Omron Sysmac Studio project Q14-16_2 (Sysmac Studio 1.23.0.14, StandardProject)

# Controller new_Controller_0: NX1P2-1040DT1 version 1.18
Task PrimaryTask (priority 4, period or condition 8000): Programa0

VAR_GLOBAL
    PP : BOOL;  (* at BuiltInIO://cpu/#0/Input_Bit_00 *)
    PM : BOOL;  (* at BuiltInIO://cpu/#0/Input_Bit_01 *)
    PR : BOOL;  (* at BuiltInIO://cpu/#0/Input_Bit_02 *)
    marcha_atras : BOOL;  (* at BuiltInIO://cpu/#0/Output_Bit_00 *)
    state : INT;
END_VAR
VAR_GLOBAL RETAIN
    rpm AT %D0 : DINT;  (* published *)
    mm_s AT %D4 : REAL;  (* published *)
END_VAR
VAR_GLOBAL
    Ch1Enable : BOOL;  (* at IOBus://unit#1/Ch1 Encoder Counter Operation Command/Ch1 Counter Enable *)
    Ch1Pulses : DINT;  (* at IOBus://unit#1/Ch1 Encoder Present Position *)
    Ch1PulseRate : UDINT;  (* at IOBus://unit#1/Ch1 Pulse Rate *)
    Ch1PeriodEnable : BOOL;  (* at IOBus://unit#1/Ch1 Pulse Period Measurement Function/Ch1 Pulse Period Measurement Enable *)
    detector_inicial : BOOL;  (* at BuiltInIO://cpu/#0/Input_Bit_03 *)
    marcha_adelante : BOOL;  (* at BuiltInIO://cpu/#0/Output_Bit_01 *)
END_VAR
VAR_GLOBAL RETAIN
    mm AT %D8 : DINT;  (* published *)
END_VAR
VAR_GLOBAL
    Ch1Reset : BOOL;  (* at IOBus://unit#1/Ch1 Encoder Counter Operation Command/Ch1 Internal Reset Execution *)
    multivelocidad_1 : BOOL;  (* at BuiltInIO://cpu/#0/Output_Bit_02 *)
    multivelocidad_2 : BOOL;  (* at BuiltInIO://cpu/#0/Output_Bit_03 *)
END_VAR
VAR_GLOBAL RETAIN
    selector_velocidad AT %D12 : INT;  (* published *)
    frecuencia_aplicada AT %D16 : INT;  (* published *)
    rpm_30hz AT %D20 : DINT;  (* published *)
    rpm_50hz AT %D24 : DINT;  (* published *)
    rpm_80hz AT %D28 : DINT;  (* published *)
    mm_s_30hz AT %D32 : REAL;  (* published *)
    mm_s_50hz AT %D36 : REAL;  (* published *)
    mm_s_80hz AT %D40 : REAL;  (* published *)
    MC_state AT %D7 : INT := 0;  (* published *)
END_VAR
VAR_GLOBAL
    PM_HMI AT %W0.00 : BOOL;  (* published *)
    PP_HMI AT %W0.01 : BOOL;  (* published *)
    PR_HMI AT %W0.02 : BOOL;  (* published *)
    PM_VAR : BOOL;
    PP_VAR : BOOL;
    PR_VAR : BOOL;
END_VAR
VAR_GLOBAL RETAIN
    deslizamiento AT %D44 : REAL;  (* published *)
END_VAR

PROGRAM Programa0
VAR CONSTANT
    time_window : INT := 500;
    encoder_resolution : INT := 8000;
END_VAR
VAR
    state : INT;
    velocidad_sincrona : REAL;
END_VAR
VAR_EXTERNAL
    Ch1Enable : BOOL;
    Ch1Pulses : DINT;
    rpm : DINT;
    Ch1PulseRate : UDINT;
    Ch1PeriodEnable : BOOL;
    PP : BOOL;
    PM : BOOL;
    detector_inicial : BOOL;
    marcha_adelante : BOOL;
    marcha_atras : BOOL;
    Ch1Reset : BOOL;
    PR : BOOL;
    mm : DINT;
    multivelocidad_1 : BOOL;
    multivelocidad_2 : BOOL;
    frecuencia_aplicada : INT;
    rpm_30hz : DINT;
    mm_s_30hz : REAL;
    rpm_50hz : DINT;
    mm_s_50hz : REAL;
    rpm_80hz : DINT;
    mm_s_80hz : REAL;
    selector_velocidad : INT;
    mm_s : REAL;
    PM_VAR : BOOL;
    PM_HMI : BOOL;
    PP_HMI : BOOL;
    PP_VAR : BOOL;
    PR_HMI : BOOL;
    PR_VAR : BOOL;
    deslizamiento : REAL;
END_VAR

(* Section calculos_encoder: ladder, written here as Structured Text *)

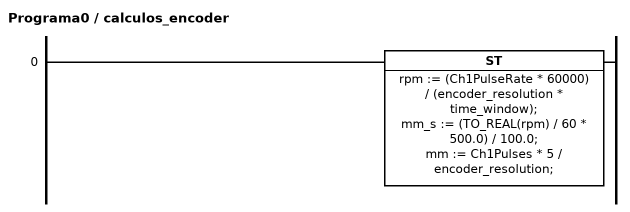
(* Rung 0 *)
rpm := (Ch1PulseRate * 60000) / (encoder_resolution * time_window);
mm_s := (TO_REAL(rpm) / 60 * 500.0) / 100.0;
mm := Ch1Pulses * 5 / encoder_resolution;

(* Section principal: ladder, written here as Structured Text *)

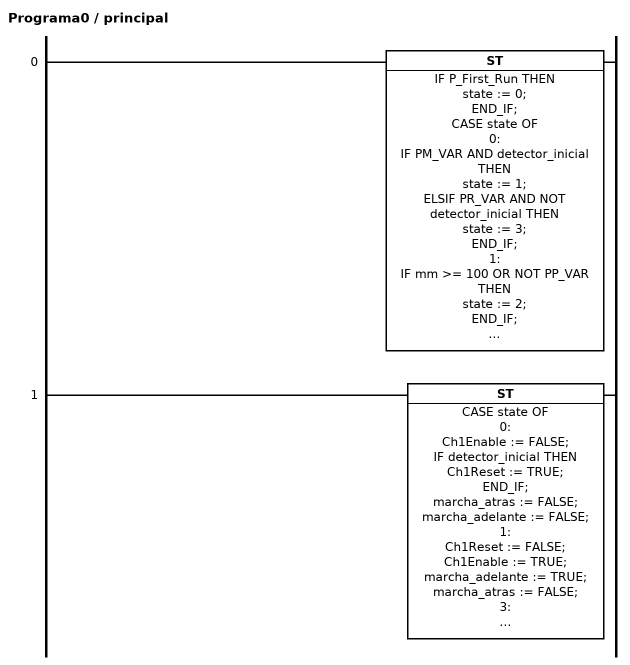
(* Rung 0 *)
IF P_First_Run THEN
    state := 0;
END_IF;

CASE state OF
    0: 
		IF PM_VAR AND detector_inicial THEN
		    state := 1;
		ELSIF PR_VAR AND NOT detector_inicial THEN
		    state := 3;
		END_IF;
	1:
		IF mm >= 100 OR NOT PP_VAR THEN
			state := 2;
		END_IF;
	2:
		IF PR_VAR THEN
			state := 3;
		END_IF;
	3:
		IF detector_inicial OR NOT PP_VAR THEN
			state := 0;
		END_IF;
END_CASE;
(* Rung 1 *)
CASE state OF
	0:
		Ch1Enable := FALSE;
		IF detector_inicial THEN
			Ch1Reset := TRUE;
		END_IF;
		marcha_atras := FALSE;
		marcha_adelante := FALSE;
	1:
		Ch1Reset := FALSE;
		Ch1Enable := TRUE;
		marcha_adelante := TRUE;
		marcha_atras := FALSE;
	3:
		Ch1Enable := TRUE;
		Ch1Reset := FALSE;
		marcha_atras := TRUE;
		marcha_adelante := FALSE;
ELSE
	Ch1Enable := TRUE;
	Ch1Reset := FALSE;
	marcha_atras := FALSE;
	marcha_adelante := FALSE;
END_CASE;

(* Section calculos_velocidad: ladder, written here as Structured Text *)

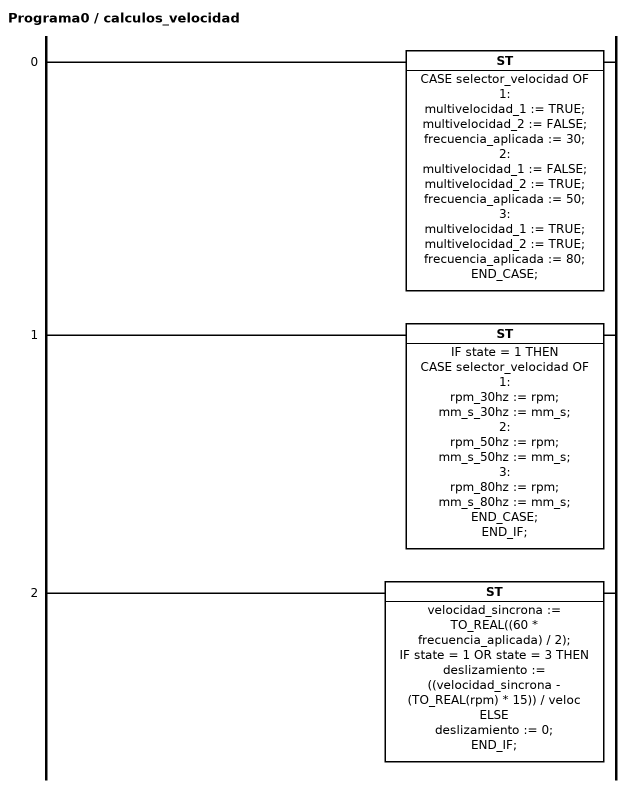
(* Rung 0 *)
CASE selector_velocidad OF
	1:
		multivelocidad_1 := TRUE;
		multivelocidad_2 := FALSE;
		frecuencia_aplicada := 30;
	2:
		multivelocidad_1 := FALSE;
		multivelocidad_2 := TRUE;
		frecuencia_aplicada := 50;
	3:
		multivelocidad_1 := TRUE;
		multivelocidad_2 := TRUE;
		frecuencia_aplicada := 80;
END_CASE;
(* Rung 1 *)
IF state = 1 THEN
	CASE selector_velocidad OF
		1:
			rpm_30hz := rpm;
			mm_s_30hz := mm_s;
		2:
			rpm_50hz := rpm;
			mm_s_50hz := mm_s;
		3:
			rpm_80hz := rpm;
			mm_s_80hz := mm_s;
	END_CASE;
END_IF;
(* Rung 2 *)
velocidad_sincrona := TO_REAL((60 * frecuencia_aplicada) / 2);

IF state = 1 OR state = 3 THEN
	deslizamiento := ((velocidad_sincrona - (TO_REAL(rpm) * 15)) / velocidad_sincrona) * 100;
ELSE
	deslizamiento := 0;
END_IF;

(* Section HMI_PLC: ladder, written here as Structured Text *)

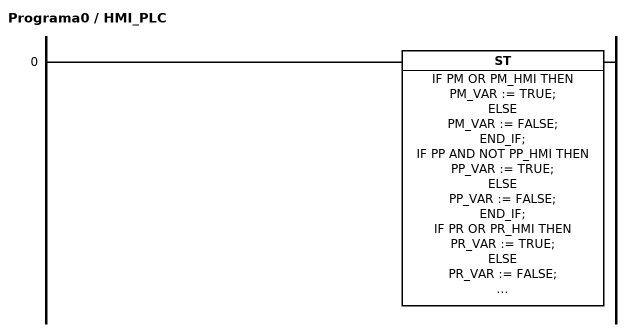
(* Rung 0 *)
IF PM OR PM_HMI THEN
	PM_VAR := TRUE;
ELSE
	PM_VAR := FALSE;
END_IF;

IF PP AND NOT PP_HMI THEN
	PP_VAR := TRUE;
ELSE
	PP_VAR := FALSE;
END_IF;

IF PR OR PR_HMI THEN
	PR_VAR := TRUE;
ELSE
	PR_VAR := FALSE;
END_IF;
END_PROGRAM